(* IEC 61131-3 sources: programs/VI-54/VI-54_20171205/VI-54_20171205/Stations/PLC_VI54/VI-54_171014/Class/StartStopPiezo, 1 file *)

(* ---- StartStopPiezo.st ---- *)
(*!
<Class
	Name               = "StartStopPiezo"
	Revision           = "3.0"
	RealtimeTask       = "false"
	CyclicTask         = "false"
	BackgroundTask     = "false"
	Sigmatek           = "false"
	OSInterface        = "false"
	HighPriority       = "false"
	Automatic          = "false"
	UpdateMode         = "Prescan"
	SharedCommandTable = "true"
	Objectsize         = "(480,300)">
	<Channels>
		<Server Name="Gestart" Visualized="false" Initialize="false" WriteProtected="true" Retentive="false"/>
		<Server Name="PiezoBediening" Visualized="true" Initialize="true" DefValue="1" WriteProtected="false" Retentive="File"/>
		<Server Name="StartNo" Visualized="false" Initialize="false" WriteProtected="false" Retentive="false"/>
		<Server Name="StopNc" Visualized="false" Initialize="false" WriteProtected="true" Retentive="false"/>
		<Client Name="iStartNo" Required="true" Internal="false"/>
		<Client Name="iStopNo" Required="true" Internal="false"/>
		<Client Name="LedGreen" Required="true" Internal="true"/>
		<Client Name="LedRed" Required="true" Internal="true"/>
		<Client Name="Merker1" Required="true" Internal="true"/>
		<Client Name="oLEDgreen" Required="false" Internal="false"/>
		<Client Name="oLEDred" Required="false" Internal="false"/>
		<Client Name="Standaard" Required="true" Internal="true"/>
	</Channels>
	<Dependencies>
		<Files>
			<File Path=".\Class\StartStopPiezo\VOV.vov"/>
		</Files>
	</Dependencies>
	<Network Name="StartStopPiezo">
		<!-- List of Components in this network -->
		<Components>
			<Object
				Name       = "LedGreen"
				Class      = "Merker"
				Position   = "(240,570)"
				Visualized = "true"
				Remotely   = "true">
				<Channels>
					<Server Name="Data"/>
				</Channels>
			</Object>
			<Object
				Name       = "LedRed"
				Class      = "Merker"
				Position   = "(240,690)"
				Visualized = "true"
				Remotely   = "true">
				<Channels>
					<Server Name="Data"/>
				</Channels>
			</Object>
			<Object
				Name       = "Merker1"
				Class      = "Merker"
				Position   = "(240,450)"
				Visualized = "true"
				Remotely   = "true">
				<Channels>
					<Server Name="Data"/>
				</Channels>
			</Object>
			<Object
				Name           = "Standaard"
				Class          = "Standard"
				Position       = "(240,270)"
				Visualized     = "false"
				BackgroundTime = "1000 ms">
				<Channels>
					<Server Name="ClassSvr"/>
				</Channels>
			</Object>
		</Components>
		<Comments>
		</Comments>
		<!-- List of Connections in this network -->
		<Connections>
			<Connection Source="this.Standaard" Destination="Standaard.ClassSvr"/>
			<Connection Source="this.Merker1" Destination="Merker1.Data"/>
			<Connection Source="this.LedGreen" Destination="LedGreen.Data"/>
			<Connection Source="this.LedRed" Destination="LedRed.Data"/>
		</Connections>
		<!-- Headerfiles -->
		<Options>
		</Options>
	</Network>
</Class>
*)
StartStopPiezo : CLASS
  //Servers:
	StartNo 	: SvrChCmd_DINT;
	StopNc 	: SvrCh_DINT;
	PiezoBediening 	: SvrCh_OptiesEnum;
	Gestart 	: SvrCh_DINT;
  //Clients:
	iStartNo 	: CltCh_DINT;
	iStopNo 	: CltCh_DINT;
	Standaard 	: CltChCmd_Standard;
	oLEDgreen 	: CltCh_DINT;
	oLEDred 	: CltCh_DINT;
	Merker1 	: CltChCmd_Merker;
	LedGreen 	: CltChCmd_Merker;
	LedRed 	: CltChCmd_Merker;
  //Variables:
		StartStatus 	: DINT;
		Signals 	: ImpClkStr;
		hStart 	: DINT;
		TmrStart 	: UDINT;
		TmrStop 	: UDINT;
		StopIntern 	: DINT;
		StartIntern 	: DINT;
  //Functions:

	FUNCTION GLOBAL StatusGestart
		VAR_INPUT
			State 	: DINT;
		END_VAR;

	FUNCTION VIRTUAL GLOBAL StartNo::Read
		VAR_OUTPUT
			output (EAX) 	: DINT;
		END_VAR;

	FUNCTION VIRTUAL GLOBAL StartNo::Write
		VAR_INPUT
			input (EAX) 	: DINT;
		END_VAR
		VAR_OUTPUT
			result (EAX) 	: DINT;
		END_VAR;

	FUNCTION VIRTUAL GLOBAL StopNc::Read
		VAR_OUTPUT
			output (EAX) 	: DINT;
		END_VAR;
  //Tables:
	FUNCTION @STD
		VAR_OUTPUT
			ret_code	: CONFSTATES;
		END_VAR;
	FUNCTION GLOBAL TAB @CT_;
END_CLASS;

#pragma using Merker
#pragma using Standard

FUNCTION VIRTUAL GLOBAL StartStopPiezo::StartNo::Read
	VAR_OUTPUT
		output (EAX) 	: DINT;
	END_VAR

  iStartNo := iStartNo.Read();
  hStart := iStartNo = 1;
  StartIntern := (Merker1.Data.Read() = 1);

  if hStart = 1 | StartIntern = 1 then
    StartNo := 1;
    TmrStart := ops.tAbsolute;
  else
    if ops.tAbsolute - TmrStart > 500 then
      StartNo := 0;
    end_if;
  end_if;
  output := StartNo;

END_FUNCTION

FUNCTION VIRTUAL GLOBAL StartStopPiezo::StopNc::Read
	VAR_OUTPUT
		output (EAX) 	: DINT;
	END_VAR

  iStopNo := iStopNo.Read();
  StopIntern := (Merker1.Data.Read() = 2);

  if PiezoBediening = Actief then
    if iStopNo = 1 | StopIntern = 1 then
      StopNc := (iStopNo = 0) & (StopIntern = 0);
      TmrStop := ops.tAbsolute;
    elsif ops.tAbsolute - TmrStop >= 400 then
      StopNc := (iStopNo = 0) & (StopIntern = 0);
    end_if;
  else
	  StopNc := (iStopNo = 1) | (StopIntern = 1);
  end_if;
  output := StopNc;

END_FUNCTION

FUNCTION GLOBAL StartStopPiezo::StatusGestart
	VAR_INPUT
		State 	: DINT;
	END_VAR

  Gestart := State;

END_FUNCTION

FUNCTION VIRTUAL GLOBAL StartStopPiezo::StartNo::Write
	VAR_INPUT
		input (EAX) 	: DINT;
	END_VAR
	VAR_OUTPUT
		result (EAX) 	: DINT;
	END_VAR

	StartStatus := input;
  Standaard.Imp_Clk(pTimeData:= #Signals);

  if PiezoBediening = Actief then
    if StartStatus = -1 then // fault
      oLEDred   := Signals._Clk500mSec;
      oLEDgreen := 0;
    elsif StartStatus = -2 then
      oLEDred   := Signals._Clk500mSec;
      oLEDgreen := Signals._Clk500mSec = 0;
    elsif StartStatus = -3 then // ExternRease
      oLEDred   := 0;
      oLEDgreen := Signals._Clk500mSec = 0;
    elsif StartStatus = -4 then // lockstate
      oLEDred   := Signals._Clk100mSec = 1;
      oLEDgreen := Signals._Clk100mSec = 1;
    elsif StartStatus = -5 then // to start position !!
      oLEDred   := Signals._Clk100mSec = 1;
      oLEDgreen := Signals._Clk500mSec = 1;
    elsif StartStatus = -6 then // Press 1x stop, Wait for cyclus
      oLEDred   := Signals._Clk100mSec = 1;
      oLEDgreen := 1;
    elsif StartStatus = 0 then // stop
      oLEDred   := 1;
      oLEDgreen := 0;
    elsif StartStatus = 1 then
      oLEDred   := 0;
      oLEDgreen := 1;
    elsif StartStatus = 2 then
      oLEDred   := 0;
      oLEDgreen := Signals._Clk100mSec;
    else
      oLEDred   := 0;
      oLEDgreen := 0;
    end_if;
  else
    oLEDred   := 0;
    oLEDgreen := 0;
  end_if;

  if IsClientConnected(#oLEDgreen) then
    oLEDgreen.Write (oLEDgreen);
    LedGreen.Data.Write(input:= oLEDgreen);
  end_if;

  if IsClientConnected(#oLEDred) then
    oLEDred.Write (oLEDred);
    LedRed.Data.Write(input:= oLEDred);
  end_if;

 	result := StartNo;

END_FUNCTION
